// Verifies that the last call to ReadTag() returned tag 0
FUNCTION INTERNAL F_CheckReadEndOfStreamTag : HRESULT
VAR_IN_OUT
    stState : ST_ParserInternalState;
END_VAR


IF stState.nLastTag <> 0 THEN
    F_CheckReadEndOfStreamTag := stState.eParserErrorCode := E_ParserErrorCode.MoreDataAvailable;
    stState.bError := TRUE;
    RETURN;
END_IF

END_FUNCTION

(* stored: Version 1.1.0.1
   POU F_CheckReadEndOfStreamTag: Id {a771decb-a4a0-4f64-89f9-523fb6ace07a}, SpecialFunc None *)
